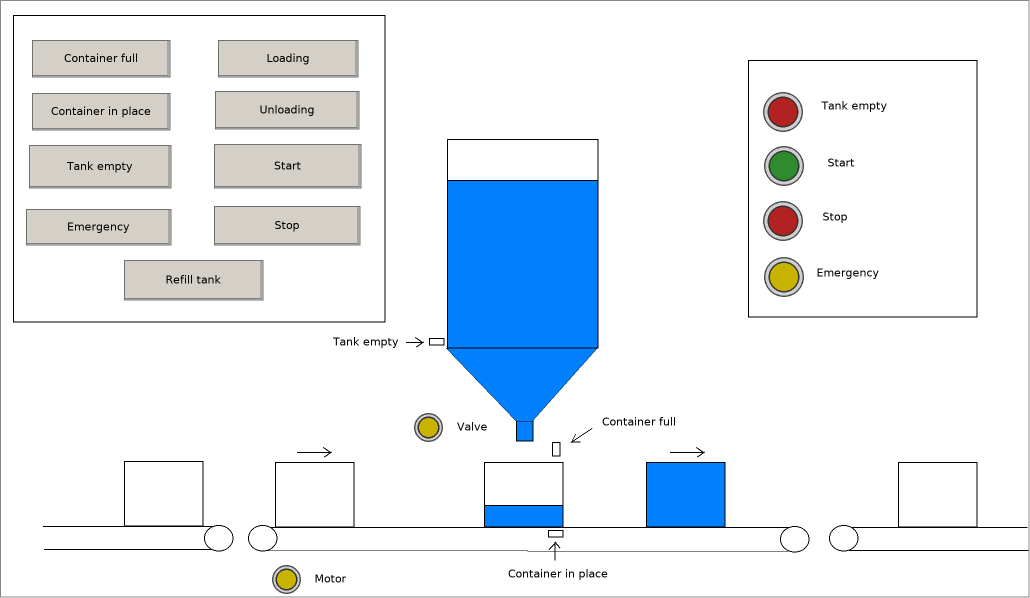
VISUALIZATION Visualization_1  // 1030x598
    Rectangle (13,15 372x307)
    Rectangle (748,60 229x257)
    Button (32,93 138x37), "Container in place", colour toggle: MAIN.Container_in_place
        toggle MAIN.Container_in_place
    Button (32,40 138x37), "Container full", colour toggle: MAIN.Container_full
        toggle MAIN.Container_full
    Button (29,145 142x43), "Tank empty", colour toggle: MAIN.Tank_empty_in
        toggle MAIN.Tank_empty_in
    Button (218,40 140x37), "Loading"
        tap MAIN.Loading
    Button (215,91 144x38), "Unloading"
        tap MAIN.Unloading
    Button (214,144 147x44), "Start", colour toggle: MAIN.Start
        toggle MAIN.Start
    Button (214,206 146x39), "Stop", colour toggle: MAIN.Stop
        toggle MAIN.Stop
    Button (26,209 145x36), "Emergency", colour toggle: MAIN.Emergency
        toggle MAIN.Emergency
    Line (43,526) (222,526)
    Line (44,549) (223,549)
    Ellipse (204,525 29x26)
    Line (256,527) (795,527)
    Line (258,550) (797,551)
    Ellipse (780,526 29x26)
    Ellipse (248,525 29x26)
    Line (848,527) (1027,527)
    Line (849,550) (1028,550)
    Ellipse (829,525 29x26)
    Rectangle (124,461 79x65)
    Rectangle (275,462 79x65), invisible if: NOT MAIN.S1
    Rectangle (484,462 79x65), invisible if: NOT MAIN.S2
    Rectangle (646,462 79x65), invisible if: NOT MAIN.S3
    Rectangle (898,462 79x65)
    Rectangle (447,139 151x209)
    Rectangle (516,420 17x21)
    Line (297,452) (331,452), invisible if: (NOT MAIN.S1) OR (MAIN.EMERGENCY)
    Line (323,447) (330,452), invisible if: (NOT MAIN.S1) OR (MAIN.EMERGENCY)
    Line (331,452) (324,457), invisible if: (NOT MAIN.S1) OR (MAIN.EMERGENCY)
    Line (670,452) (704,452), invisible if: (NOT MAIN.S3) OR (MAIN.EMERGENCY)
    Line (696,447) (703,452), invisible if: (NOT MAIN.S3) OR (MAIN.EMERGENCY)
    Line (704,452) (697,457), invisible if: (NOT MAIN.S3) OR (MAIN.EMERGENCY)
    Line (406,342) (423,342)
    Line (415,337) (422,342)
    Line (423,342) (416,347)
    Line (555,560) (555,542)
    Line (549,549) (555,543)
    Line (560,548) (555,542)
    Rectangle (429,338 15x7)
    Rectangle (548,530 15x7)
    Rectangle (552,442 8x14)
    Line (571,442) (592,428)
    Line (575,434) (571,442)
    Line (580,442) (572,442)
    Lamp1 (760,84 46x56), variable: MAIN.Tank_empty_out, style: Lamp-Lamp1-Red
    Label (812,91 85x30), "Tank empty"
    Lamp1 (761,138 46x56), variable: MAIN.Start, style: Lamp-Lamp1-Green
    Lamp1 (760,193 46x56), variable: MAIN.Stop, style: Lamp-Lamp1-Red
    Label (481,552 154x44), "Container in place"
    Label (289,320 154x44), "Tank empty"
    Label (562,400 154x44), "Container full"
    Rectangle (447,180 151x168), invisible if: MAIN.Tank_empty_in
    Rectangle (516,420 17x21), invisible if: MAIN.Tank_empty_in
    Rectangle (484,505 79x22), invisible if: NOT MAIN.S2
    Label (817,148 48x30), "Start"
    Label (809,202 52x30), "Stop"
    Lamp1 (270,563 33x33), variable: MAIN.Motor, style: Lamp-Lamp1-Yellow
    Label (303,564 55x30), "Motor"
    Lamp1 (412,411 33x33), variable: MAIN.Valve, style: Lamp-Lamp1-Yellow
    Label (445,412 55x30), "Valve"
    Lamp1 (761,249 46x56), variable: MAIN.Emergency, style: Lamp-Lamp1-Yellow
    Label (807,258 82x30), "Emergency"
    Button (124,260 139x40), "Refill tank"
        tap MAIN.Refill
    Polygon (446,348) (523,348) (597,348) (532,421) (516,421), colour toggle: MAIN.Tank_empty_in
END_VISUALIZATION

(* stored: Version 1.1.0.1, ProductVersion 3.1.4020.6
   Visu Visualization_1: Id {4517b380-3f05-4c5a-bb5a-903988fcf258} *)
